FUNCTION F_Convert_2Byte_to_Uint 

VAR_IN_OUT
	inputNum : UINT; 
	dataByte1 : BYTE;
	dataByte2 : BYTE;
END_VAR

VAR
	arrByte : ARRAY [0..1] OF BYTE;
END_VAR

arrByte[0]:= dataByte1;
arrByte[1]:= dataByte2;
MEMCPY(ADR(inputNum), ADR(arrByte), 2);

//F_Convert_Int_to_2Byte:=arrByte;

END_FUNCTION

(* stored: Version 1.1.0.1, ProductVersion 3.1.4024.11
   POU F_Convert_2Byte_to_Uint: Id {29a40994-dd29-4b3e-b5d3-5fbe007c0cab}, SpecialFunc None *)
